FUNCTION_BLOCK FB_Sensor
VAR_INPUT
	stIn				:	ST_CSL_In;
	bEnable				:	BOOL;
	
END_VAR

VAR_OUTPUT
	eStep				:	E_Step;
	eErrStep			:	E_Step;
	nErrId				:	DINT;
	tStepTime			:	TIME;
	
	bFbEnd				:	BOOL;
	
	stOut				:	ST_CSL_RawOut;
	
	nSlot				:	INT;
	
END_VAR

VAR_IN_OUT
	
END_VAR

VAR
	bInitialized		:	BOOL;
	eNewStep			:	E_Step;
	bEntryAct			:	BOOL;
	fbTonStart			:	TON;
	
	fbMeasure			:	FB_Measuring;
	fbSlot				:	FB_Processing;
	
	stParams			:	ST_CSL_Params;
	
	rPieceValue			:	REAL;
	bEndMeasure			:	BOOL;
	
END_VAR

(*Initialization of the FB_Sensor*)
IF NOT bInitialized THEN
	eNewStep := E_Step.NoStep;
	eStep := E_Step.Start;
	bEntryAct := FALSE;
	bFbEnd := FALSE;
	bInitialized := TRUE;
ELSE
	
	(*Preamble*)
	
	(*Forcing the Error State*)
	IF NOT bEnable THEN
		eNewStep := E_Step.NeOrError;
	END_IF	
	
	(*State change management*)
	IF eNewStep <> E_Step.NoStep THEN
		eStep := eNewStep;
		eNewStep := E_Step.NoStep;
		bEntryact := FALSE;
	END_IF
	
	(*Filters*)
	fbTonStart(IN := stIn.bPieceSensorInput, PT := T#2S);
	
	
	(*Case*)
	CASE eStep OF
		(*Start Step*)
		E_Step.Start :
			(*Body*)
			stOut.bLStart	:= TRUE;
			stOut.bLStop := FALSE;
			stOut.bLAck := FALSE;
			
			stOut.bMotor := FALSE;
		
			(*Transition - to Measuring*)
			IF fbTonStart.Q AND bEnable THEN
				eNewStep := E_Step.Measuring;
			END_IF
			
			(*Exit Act*)
			IF eNewStep <> E_Step.NoStep THEN
				IF eNewStep = E_Step.NeOrError THEN
					eErrStep := eStep;
					//nErrId	:= 16#9999_9999;
				END_IF
			END_IF
			
		(*Measuring Step*)
		E_Step.Measuring :
			(*Body*)
			stOut.bLStart	:= TRUE;
			stOut.bLStop := FALSE;
			stOut.bLAck := FALSE;
			
			stOut.bMotor := TRUE;
		
			fbMeasure(Vin := stIn.nColorSensor, Vout := rPieceValue);
			
			(*Transition - to Processing*)
			IF fbMeasure.EndMeasure AND bEnable THEN
				eNewStep := E_Step.Processing;
			END_IF
			
			(*Exit Act*)
			IF eNewStep <> E_Step.NoStep THEN
				IF eNewStep = E_Step.NeOrError THEN
					eErrStep := eStep;
					//nErrId	:= 16#9999_9999;
				END_IF
			END_IF
			
		(*Processing Step*)
		E_Step.Processing :
			(*Body*)
			stOut.bLStart := TRUE;
			stOut.bLStop := FALSE;
			stOut.bLAck := FALSE;

			stOut.bMotor := TRUE;
			
			fbSlot(SensorInput := rPieceValue, stParams := stParams);
			nSlot := fbSlot.slot;
			
			(*Transition - to exit*)
			IF fbTonStart.Q AND bEnable THEN
				bInitialized := FALSE;
				bFbEnd := TRUE;
			END_IF
			
			(*Exit Act*)
			IF eNewStep <> E_Step.NoStep THEN
				IF eNewStep = E_Step.NeOrError THEN
					eErrStep := eStep;
					//nErrId	:= 16#9999_9999;
				END_IF
			END_IF
	END_CASE
END_IF

END_FUNCTION_BLOCK

(* stored: Version 1.1.0.1, ProductVersion 3.1.4024.12
   POU FB_Sensor: Id {9fa85518-2ab9-47fc-a442-bf72b57e6579}, SpecialFunc None *)
